FUNCTION_BLOCK CLIENT_0_4 (* 4-Output Client Interface *)
  (* Standard: 61499-1; Classification: Communications *)
  (* Version 1.0, 21-03-12, GASR, Universidade do Estado de Santa Catarina *)
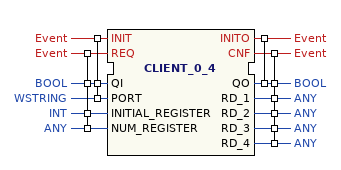
  EVENT_INPUT
    INIT WITH QI, PORT; (* Service Initialization *)
    REQ WITH QI, INITIAL_REGISTER, NUM_REGISTER; (* Service Request *)
  END_EVENT
  EVENT_OUTPUT
    INITO WITH QO; (* Initialization Confirm *)
    CNF WITH QO, RD_1, RD_2, RD_3, RD_4; (* Service Confirmation *)
  END_EVENT
  VAR_INPUT
    QI : BOOL; (* Event Input Qualifier *)
    PORT : WSTRING; (* Connection Identifier *)
    INITIAL_REGISTER : INT; (* Value of the initial register *)
    NUM_REGISTER : ANY; (* Data to Send *)
  END_VAR
  VAR_OUTPUT
    QO : BOOL; (* Event Output Qualifier *)
    RD_1 : ANY; (* Received Data *)
    RD_2 : ANY; (* Received Data *)
    RD_3 : ANY; (* Received Data *)
    RD_4 : ANY; (* Received Data *)
  END_VAR
END_FUNCTION_BLOCK
